FUNCTION_BLOCK ZAppSequenceBoot EXTENDS ZAppSequence IMPLEMENTS ZCore.ISequence
VAR
  _step : ZCore.Step(ZAppStep.BootBegin, ZAppStep.BootEnd);
END_VAR

IF OnStart(_step)
THEN
  // init custom sequence variables here ...
END_IF

REPEAT
  LogStep();

  CASE _step.Index OF
    (* -------------------------------------------------------------------------------------------------------------------------------- *)
    ZAppStep.BootBegin:
    (* -------------------------------------------------------------------------------------------------------------------------------- *)
    
      IF _step.OnEntry()
      THEN
        ZModuleProgram.SetLoggerLevel(ZCore.LogLevel.Trace);
        ZModuleProgram.Logger.AddLogger(ZModuleProgram.LoggerFile);        
        {attribute '__ZwPlcAppZComModuleContext__'} // Do not remove this attribute! It is used for code generation.      
      END_IF
      
	  IF ZModuleProgram.Datetime.State <> ZCore.ObjectState.Booting
      THEN
        _step.SetNext(ZAppStep.BootLoadDefaultData);        
      END_IF
      
    (* -------------------------------------------------------------------------------------------------------------------------------- *)
    ZAppStep.BootLoadDefaultData:
    (* -------------------------------------------------------------------------------------------------------------------------------- *)

      {warning 'The application is loading the default config data on every restart!'}
      LoadDefaultConfigData();
      
      IF IsCommissioning()
      THEN
        LoadDefaultData();
      END_IF
      
      _step.SetNext(ZAppStep.BootEnd);
      
    (* -------------------------------------------------------------------------------------------------------------------------------- *)
    ZAppStep.BootEnd:
    (* -------------------------------------------------------------------------------------------------------------------------------- *)
      SetBusy(FALSE);
      
  ELSE
    Abort('sequence contains unhandled step');
  END_CASE
UNTIL _step.IsNotRepeatable() OR_ELSE NOT Busy END_REPEAT

METHOD  IsCommissioning : BOOL
IsCommissioning := TRUE;
END_METHOD

METHOD FINAL LoadDefaultConfigData

{region "Transport"}
  {IF NOT (defined (Transport_disabled))}
  ZGlobal.Data.Config.Transport.Simulated := TRUE;
  {region "UserInitCode"}
  // put your individual init code for this unit here
  ZGlobal.Data.Machine.Transport.Highspeed := 10.0;
  ZGlobal.Data.Machine.Transport.Slowspeed := 2.0;
        
  ZGlobal.Data.Machine.Transport.HorizontalLeftPos := 2.0;
  ZGlobal.Data.Machine.Transport.HorizontalRightPos := 8.0;
  ZGlobal.Data.Machine.Transport.HorizontalHomePos := 0.0;
        
  ZGlobal.Data.Machine.Transport.VerticalBottomPos := 5.0;
  ZGlobal.Data.Machine.Transport.VerticalTopPos := 2.0;
  ZGlobal.Data.Machine.Transport.VerticalHomePos := 0.0;
  {endregion}
  {END_IF}
  {attribute 'ZId' := '413070d6-61de-4759-aae5-e3ab76278fe1'}
{endregion}

{region "Drilling"}
  {IF NOT (defined (Drilling_disabled))}
  ZGlobal.Data.Config.Drilling.Simulated := TRUE;
  {region "UserInitCode"}
  // put your individual init code for this unit here
  {endregion}
  {END_IF}
  {attribute 'ZId' := 'a0f6f6d1-15cf-44f1-8585-ff8bdaab6c0e'}
{endregion}

{region "Assembly"}
  {IF NOT (defined (Assembly_disabled))}
  ZGlobal.Data.Config.Assembly.Simulated := TRUE;
  {region "UserInitCode"}
  // put your individual init code for this unit here
  {endregion}
  {END_IF}
  {attribute 'ZId' := 'fe48c71e-df5c-4f02-81a6-6f01ddca37c0'}
{endregion}

{region "QualityInspection"}
  {IF NOT (defined (QualityInspection_disabled))}
  ZGlobal.Data.Config.QualityInspection.Simulated := TRUE;
  {region "UserInitCode"}
  // put your individual init code for this unit here
  {endregion}
  {END_IF}
  {attribute 'ZId' := 'a1721ee9-e163-4dba-818e-d45d6db51cc5'}
{endregion}

{attribute '__ZwPlcUnitLoadDefaultConfigData__'} // Do not remove this attribute! It is used for code generation.
END_METHOD

METHOD FINAL LoadDefaultData

{attribute '__ZwPlcUnitLoadDefaultData__'} // Do not remove this attribute! It is used for code generation.
END_METHOD

END_FUNCTION_BLOCK

(* stored: Version 1.1.0.1
   POU ZAppSequenceBoot: Id {ac255339-67bc-40f5-86b7-534b88d2ae0e}, SpecialFunc None
   Method IsCommissioning: Id {a3ea03ec-ee5f-4d37-b289-be135ee49366}
   Method LoadDefaultConfigData: Id {033f4bff-60a4-468c-8813-fef0ea28cd35}
   Method LoadDefaultData: Id {fa9633c4-76dc-4ebb-990b-7115ef78f212} *)
